{attribute 'linkalways'} 
{attribute 'no_explicit_call' := 'This FB is a CLASS and must be accessed using methods or properties'}
{attribute 'enable_dynamic_creation'}
FUNCTION_BLOCK InputPortAddedEvent EXTENDS Disposable IMPLEMENTS I_InputPortAddedEvent
VAR
	_targetInputPort : I_InputPort;
END_VAR

METHOD FB_init : BOOL
VAR_INPUT
	bInitRetains : BOOL; // if TRUE, the retain variables are initialized (warm start / cold start)
	bInCopyCode : BOOL;  // if TRUE, the instance afterwards gets moved into the copy code (online change)
	TargetInputPort : I_InputPort;
END_VAR
This^._targetInputPort := TargetInputPort;
END_METHOD

PROPERTY PUBLIC TargetInputPort : I_InputPort
GET
TargetInputPort := _targetInputPort;
END_GET
END_PROPERTY

END_FUNCTION_BLOCK

(* stored: Version 1.1.0.1, ProductVersion 3.1.4024.12
   POU InputPortAddedEvent: Id {87da74a1-1f3b-0af2-0856-b01263bc7284}, SpecialFunc None
   Folder Constructor: Id {4b92a883-34c7-0ffb-1558-d7c9b68d5fee}
   Method FB_init: Id {5203ab3a-4271-04c9-3be5-e45e64613c28}
   Property TargetInputPort: Id {5190413e-9637-0cff-1a5e-9b71d3ecc836}
   Get Get: Id {047a7663-b306-07a4-07d9-ef1edc5c8780} *)
